(* PLC project Unnamed, Unknown Unnamed 1 *)
(* stored: creationDateTime 2023-09-18T19:23:44, modificationDateTime 2023-09-19T10:05:35 *)

PROGRAM program0
  VAR_IN_OUT
    StartButton : BOOL;
    RollerEngine : BOOL;
    Nozzle : BOOL;
    BottleSensor : BOOL;
    WaterLevelSensor : BOOL;
    PlantState : INT;
  END_VAR

            (* Initialization Phase*)
    IF PlantState = 0 THEN
        RollerEngine := FALSE;
        Nozzle := FALSE;
        IF StartButton THEN
            PlantState := 1;         (* Move to Filling Phase*)
        END_IF;
    END_IF;

    (*Filling Phase*)
    IF PlantState = 1 THEN
        IF BottleSensor AND NOT WaterLevelSensor THEN
            Nozzle := TRUE;         (*Open the nozzle if bottle is under and not filled*)
        ELSE
            Nozzle := FALSE;        (* Close the nozzle otherwise*)
        END_IF;

        IF WaterLevelSensor THEN
            PlantState := 2;        (*Move to Moving Phase once bottle is filled*)
        END_IF;
    END_IF;

    (*Moving Phase*)
    IF PlantState = 2 THEN
        Nozzle := FALSE;            (* Ensure nozzle is closed*)
        RollerEngine := TRUE;        (* Start the roller engine to move the bottle*)

        IF NOT BottleSensor THEN
            PlantState := 1;         (*Move back to Filling Phase once bottle has moved away*)
        END_IF;
    END_IF;

  (* Stop the plant if StartButton is turned off*)
    IF NOT StartButton THEN
        PlantState := 0;
    END_IF;
          
END_PROGRAM

CONFIGURATION Config0
  RESOURCE Res0 ON PLC
    TASK task0(INTERVAL := T#20ms, PRIORITY := 0);
    PROGRAM instance0 WITH task0 : program0;
  END_RESOURCE
END_CONFIGURATION
